// TIA Portal V17 export
// export: Created 2022-07-28T18:03:20.7885724Z, ExportSetting None, DisplayName Totally Integrated Automation Portal, DisplayVersion V17, DisplayName TIA Portal Openness, DisplayVersion V17, DisplayName TIA Portal Teamcenter Gateway, DisplayVersion V17, DisplayName TIA Portal Version Control Interface, DisplayVersion V17, DisplayName TIA Portal Test Suite Advanced, DisplayVersion V17, DisplayName SINAMICS Startdrive Advanced, DisplayVersion V17, DisplayName SINAMICS DCC, DisplayVersion V17, DisplayName SINAMICS Startdrive G130, G150, S120, S150, SINAMICS MV, S210, DisplayVersion V17, DisplayName SINAMICS Startdrive G110M, G120, G120C, G120D, G120P, G115D, DisplayVersion V17, DisplayName STEP 7 Professional, DisplayVersion V17, DisplayName SIMATIC Energy Suite, DisplayVersion V17, DisplayName STEP 7 CFC, DisplayVersion V17, DisplayName STEP 7 Safety, DisplayVersion V17, DisplayName WinCC Advanced / Unified PC, DisplayVersion V17, DisplayName SIMATIC Visualization Architect, DisplayVersion V17
TYPE "_SlideGate_Pneumo_Counters"
   STRUCT
      di_TimeOper_Tot { ExternalWritable := 'False'; S7_SetPoint := 'True'} : DInt;   // Total Time Operating time in hours
      di_Activ_tot { ExternalWritable := 'False'; S7_SetPoint := 'True'} : DInt;   // Counter object activated switches/switching operations
   END_STRUCT;
END_TYPE
